FUNCTION_BLOCK FB_Inverter_Sim IMPLEMENTS I_Inverter
VAR_INPUT
END_VAR
VAR_OUTPUT
END_VAR
VAR
	TargetSpeed			: REAL;
	fActualSpeed 		: REAL;
	bBrake 		  		: BOOL;
	nErrId				: INT;
	bExecute 			: BOOL;
	bStop				: BOOL;
	bReset				: BOOL;
	//Var sim
	nState				: INT;
	tTimer				: TON;
	tDelay				: TIME := T#2000MS; //acceleration time of inverter
	bStopInit			: BOOL := TRUE;
	fTargetSpeed_re1	: REAL;
	fTargetSpeed_re2	: REAL;
	fActualSpeed_re		: REAL;
END_VAR

CASE nState OF
	0: //init set stop inverter
		IF bStopInit THEN
			bStop := TRUE;
			fActualSpeed := 0;
			tTimer(IN := FALSE);
		END_IF
		nState := nState + 1;
	1://Inv Stop
		fActualSpeed := 0;
		tTimer(IN := FALSE);
		
	10://Inv Run after bExecute = true and speed <> 0
		tTimer(IN := TRUE,PT := tDelay);
		fActualSpeed := fActualSpeed_re + (TIME_TO_REAL(tTimer.ET)*(fTargetSpeed_re1/TIME_TO_REAL(tDelay)));
		fInvSpeed := fActualSpeed;
		// check when change targetspeed
		IF fTargetSpeed_re2 < fTargetSpeed OR fTargetSpeed_re2 > fTargetSpeed THEN
			nState := 20;
		END_IF
	20:
		fActualSpeed_re := fActualSpeed;
		fTargetSpeed_re1 := fTargetSpeed - fActualSpeed;
		fTargetSpeed_re2 := fTargetSpeed;
		tTimer(IN := FALSE);
		nState := 10;
		
END_CASE

//check for signal
IF bExecute AND (fTargetSpeed <> 0) AND (nState = 1) THEN
	fTargetSpeed_re1 := fTargetSpeed;
	fTargetSpeed_re2 := fTargetSpeed;
	fActualSpeed_re := fActualSpeed;
	tTimer(IN := FALSE);
	nState := 10;//Inv run
END_IF

IF bStop THEN
	fActualSpeed := 0;
	nState := 1;//
END_IF

IF fActualSpeed = 0 THEN
	bHaveLoad := FALSE;
ELSE
	bHaveLoad := TRUE;
END_IF

PROPERTY ActualSpeed : REAL
GET
ActualSpeed := fActualSpeed/100;
END_GET
END_PROPERTY

PROPERTY bIsMove : BOOL
GET
IF ActualSpeed > 3 THEN
	bIsMove := FALSE;
ELSE
	bIsMove := TRUE;
END_IF
END_GET
END_PROPERTY

PROPERTY fTargetSpeed : REAL
GET
fTargetSpeed := TargetSpeed;
END_GET
SET
TargetSpeed := fTargetSpeed;
END_SET
END_PROPERTY

METHOD Reset : BOOL
VAR_INPUT
END_VAR
bExecute := FALSE;
bStop	 := FALSE;
bReset	 := TRUE;
END_METHOD

METHOD Reverse : BOOL
VAR_INPUT
END_VAR
END_METHOD

METHOD Start : BOOL
VAR_INPUT
END_VAR
bExecute := TRUE;
bStop	 := FALSE;
bReset	 := FALSE;
END_METHOD

METHOD Stop : BOOL
VAR_INPUT
END_VAR
bExecute := FALSE;
bStop	 := TRUE;
bReset	 := FALSE;
END_METHOD

END_FUNCTION_BLOCK

(* stored: Version 1.1.0.1, ProductVersion 3.1.4024.12
   POU FB_Inverter_Sim: Id {defff990-0e79-45e4-92d8-f76780ecb9c9}, SpecialFunc None
   Property ActualSpeed: Id {43e3d9a2-9d79-4976-a463-fa505267646b}
   Get Get: Id {ed6323ac-0d4f-4356-85b4-e47aad09a4ac}
   Property bIsMove: Id {bb52d2c6-1caf-4581-8604-f5b5a52b9a58}
   Get Get: Id {0ce38896-a388-4159-9bce-f8397caabb4d}
   Property fTargetSpeed: Id {589223b5-93a4-4695-8fa1-a94425e1dfdb}
   Get Get: Id {006632f1-4fd8-4298-888a-ec89b89edcce}
   Set Set: Id {43691246-d78a-4ec3-8c20-673b043bf8a0}
   Method Reset: Id {69a1fd62-8424-4d9e-8633-8c5bfff97448}
   Method Reverse: Id {d78c5eaf-a0df-4ad9-bb14-98c385aaeb63}
   Method Start: Id {3cdeaf80-1c64-42f4-8ca6-49981d396e36}
   Method Stop: Id {1f25b007-8c9d-4ffd-a5e2-fefa14b6d500} *)
